FUNCTION exF_POWER : REAL
VAR_INPUT
	a: REAL;
	x: REAL;
	n: REAL;
END_VAR

exF_POWER := a * EXPT(X, N);

END_FUNCTION

(* stored: Version 1.1.0.1, ProductVersion 3.1.4024.3
   POU exF_POWER: Id {630ecc23-a5d9-4c92-886f-959580e94731}, SpecialFunc None *)
